FUNCTION_BLOCK FB_Valve_Ctrl
VAR_INPUT
	i_Interlocks		:ARRAY[1..5] OF BOOL;
	i_ProcesslocksOK	:BOOL;
	i_AutoCmd			:BOOL;
	i_ManCmd			:BOOL;
	i_ServiceMode		:BOOL;
	i_EnableHP			:BOOL;
	i_EnableWP			:BOOL;
	i_HP				:BOOL;
	i_WP				:BOOL;
	i_Timeout			:TIME;
END_VAR
VAR_OUTPUT
	q_InterlocksOK		:BOOL;
	q_bEnabled			:BOOL;
	q_bCmd				:BOOL;
	q_bHP				:BOOL;
	q_bWP				:BOOL;
	q_bTraveling		:BOOL;
	q_bHP_Timeout		:BOOL;
	q_bWP_Timeout		:BOOL;
	q_cmd_Timeout		:BOOL;
	q_Faulted			:BOOL;
END_VAR
VAR
	tonTimeoutHP		:TON;
	tonTimeoutWP		:TON;
	tonTimeoutCmd		:TON;
	tofDelayOut			:TOF;
	bCmd				:BOOL;
END_VAR

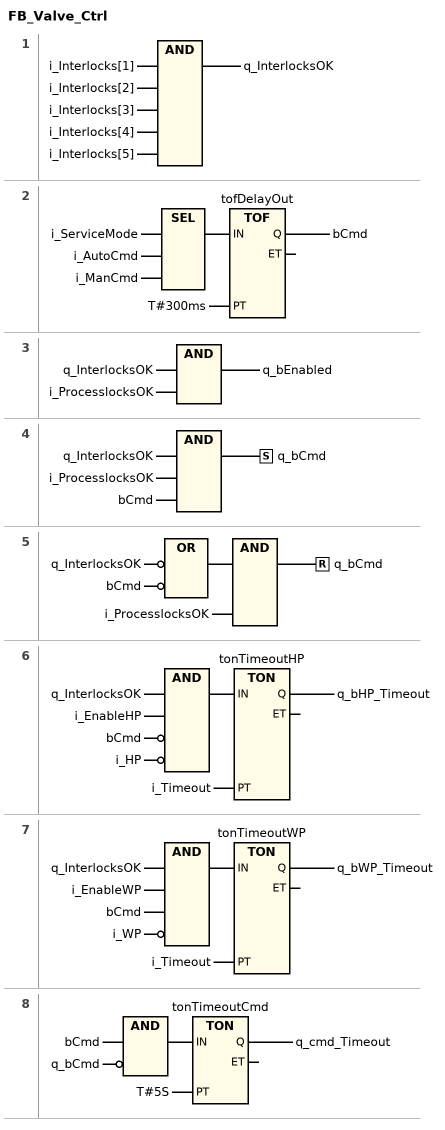
// NETWORK 1
q_InterlocksOK := i_Interlocks[1] AND i_Interlocks[2] AND i_Interlocks[3] AND i_Interlocks[4] AND i_Interlocks[5];

// NETWORK 2
tofDelayOut(IN := SEL(i_ServiceMode, i_AutoCmd, i_ManCmd), PT := T#300ms); // TOF
bCmd := tofDelayOut.Q;

// NETWORK 3
q_bEnabled := q_InterlocksOK AND i_ProcesslocksOK;

// NETWORK 4
q_bCmd S= q_InterlocksOK AND i_ProcesslocksOK AND bCmd;

// NETWORK 5
q_bCmd R= (NOT q_InterlocksOK OR NOT bCmd) AND i_ProcesslocksOK;

// NETWORK 6
tonTimeoutHP(IN := q_InterlocksOK AND i_EnableHP AND NOT bCmd AND NOT i_HP, PT := i_Timeout); // TON
q_bHP_Timeout := tonTimeoutHP.Q;

// NETWORK 7
tonTimeoutWP(IN := q_InterlocksOK AND i_EnableWP AND bCmd AND NOT i_WP, PT := i_Timeout); // TON
q_bWP_Timeout := tonTimeoutWP.Q;

// NETWORK 8
tonTimeoutCmd(IN := bCmd AND NOT q_bCmd, PT := T#5S); // TON
q_cmd_Timeout := tonTimeoutCmd.Q;

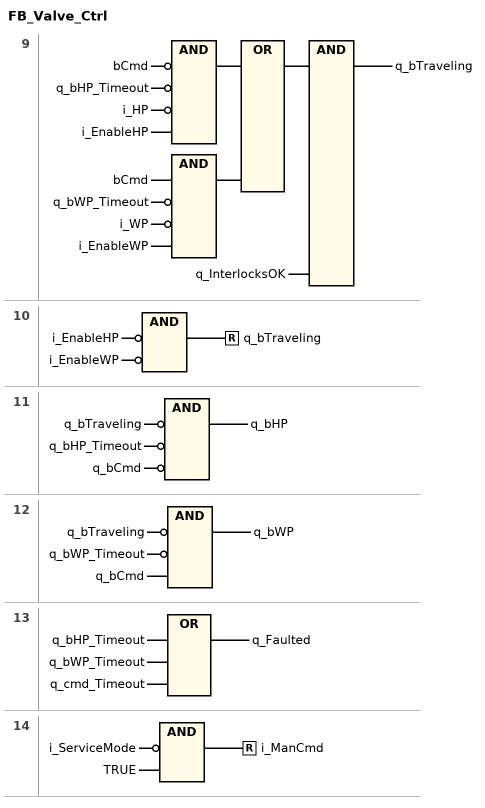
// NETWORK 9
q_bTraveling := (NOT bCmd AND NOT q_bHP_Timeout AND NOT i_HP AND i_EnableHP OR bCmd AND NOT q_bWP_Timeout AND NOT i_WP AND i_EnableWP) AND q_InterlocksOK;

// NETWORK 10
q_bTraveling R= NOT i_EnableHP AND NOT i_EnableWP;

// NETWORK 11
q_bHP := NOT q_bTraveling AND NOT q_bHP_Timeout AND NOT q_bCmd;

// NETWORK 12
q_bWP := NOT q_bTraveling AND NOT q_bWP_Timeout AND q_bCmd;

// NETWORK 13
q_Faulted := q_bHP_Timeout OR q_bWP_Timeout OR q_cmd_Timeout;

// NETWORK 14
i_ManCmd R= NOT i_ServiceMode AND TRUE;

END_FUNCTION_BLOCK

(* stored: Version 1.1.0.1, ProductVersion 3.1.4024.12
   POU FB_Valve_Ctrl: Id {91ca9d7f-f66d-41d6-8060-5a489d3e2135}, SpecialFunc None *)
